PROGRAM main
VAR
	GreenOn : bool := True;
	AllLightsOff : bool := False;
	YellowOn : bool := False;
	RedOn : bool := False;
	GreenTimer : TON;
	YellowTimer : TON;
	RedTimer : TON;
END_VAR

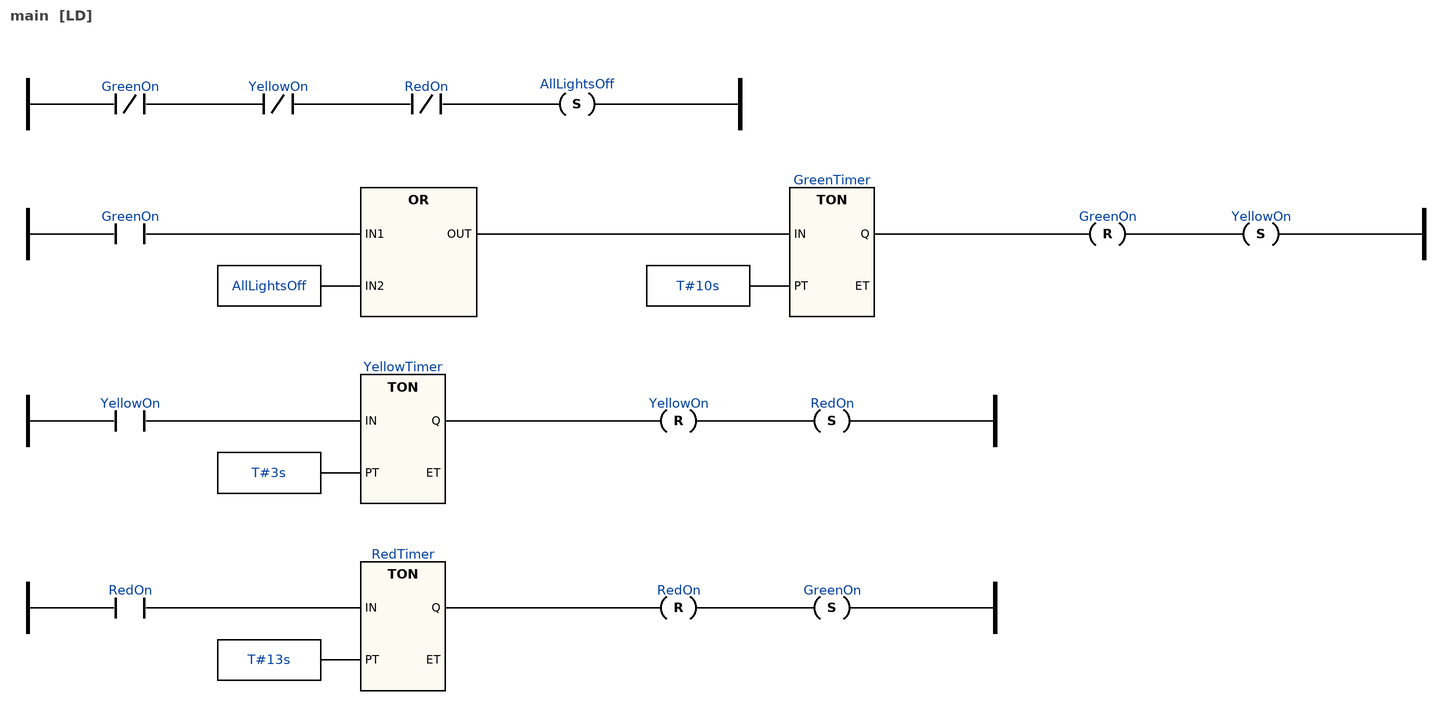
(* LD diagram, written out as Structured Text *)
IF NOT GreenOn AND NOT YellowOn AND NOT RedOn THEN AllLightsOff := TRUE; END_IF;
GreenTimer(IN := GreenOn OR AllLightsOff, PT := T#10s);
IF GreenTimer.Q THEN GreenOn := FALSE; END_IF;
IF GreenTimer.Q THEN YellowOn := TRUE; END_IF;
YellowTimer(IN := YellowOn, PT := T#3s);
IF YellowTimer.Q THEN YellowOn := FALSE; END_IF;
IF YellowTimer.Q THEN RedOn := TRUE; END_IF;
RedTimer(IN := RedOn, PT := T#13s);
IF RedTimer.Q THEN RedOn := FALSE; END_IF;
IF RedTimer.Q THEN GreenOn := TRUE; END_IF;
END_PROGRAM
